// TIA Portal project "code_V15.1" (V15.1)

(* hardware
DEVICE "S7-1200 station_1"  S7-1200 Station
   slot 0: "Rack_0"  S7-1200 Rack  Rack  V1.0
   slot 1: "PLC_1"  CPU 1212C AC/DC/Rly  6ES7 212-1BE40-0XB0  V4.2
DEVICE "PC-System_1"  SIMATIC PC station
   slot 0: "SIMATIC PC station"  Rail  SIMATIC PC-Station  V1.0
      slot 125: "Stationmanager"  Station_Manager  V6.0.4
   slot 1: "HMI_RT_1"  WinCC RT Advanced  6AV2 104-0xxxx-xxxx  15.0.0.0
      slot 33792: "Host interface"  Host interface
   slot 2: "IE general_1"  IE General  IE_CP  V8.2.0
*)

// ===== PLC "PLC_1"  CPU 1212C AC/DC/Rly =====

VAR_GLOBAL   // PLC tag table "INPUT"
   "start" AT %M0.0 : Bool;
   "vatDo" AT %M0.1 : Bool;
   "vatXanh" AT %M0.2 : Bool;
   "CB1" AT %M0.3 : Bool;
   "reset" AT %M0.4 : Bool;
   "bd" AT %M0.5 : Bool;
END_VAR

VAR_GLOBAL   // PLC tag table "OUTPUT"
   "soVatDo" AT %MW100 : Int;
   "soVatXanh" AT %MW102 : Int;
   "vatDoDiChuyen" AT %MW104 : Int;
   "vatXanhDiChuyen" AT %MW106 : Int;
   "demmaudo" AT %MW116 : Int;
   "demmauxanh" AT %MW118 : Int;
END_VAR

VAR_GLOBAL   // PLC tag table "TG"
   "tg1" AT %M50.0 : Bool;
   "tg2" AT %M50.1 : Bool;
   "tg3" AT %M50.2 : Bool;
   "tg4" AT %M50.3 : Bool;
   "tg5" AT %M50.4 : Bool;
   "tg6" AT %M50.5 : Bool;
   "tg7" AT %M50.6 : Bool;
   "tg8" AT %M50.7 : Bool;
   "vatdodi" AT %M51.0 : Bool;
   "vatxanhdi" AT %M51.1 : Bool;
   "tg11" AT %M51.2 : Bool;
   "tg12" AT %M51.3 : Bool;
   "tg13" AT %M51.4 : Bool;
   "tg14" AT %M51.5 : Bool;
   "tg15" AT %M51.6 : Bool;
   "tg16" AT %M51.7 : Bool;
   "tg17" AT %M52.0 : Bool;
   "tg18" AT %Q0.0 : Bool;
   "tg19" AT %M52.2 : Bool;
   "tg20" AT %M52.3 : Bool;
   "tg21" AT %M52.4 : Bool;
   "tg22" AT %M52.5 : Bool;
   "tg23" AT %M52.6 : Bool;
   "tg24" AT %M52.7 : Bool;
   "tg25" AT %M53.0 : Bool;
   "TG_star" AT %M49.7 : Bool;
   "xung1" AT %M53.1 : Bool;
   "xung2" AT %M53.2 : Bool;
   "xung3" AT %M53.3 : Bool;
   "xung4" AT %M53.4 : Bool;
   "xung5" AT %M53.5 : Bool;
   "xung6" AT %M53.6 : Bool;
   "xung7" AT %M53.7 : Bool;
   "xung8" AT %M54.0 : Bool;
   "xung9" AT %M54.1 : Bool;
   "xung10" AT %M54.2 : Bool;
END_VAR

VAR_GLOBAL   // PLC tag table "TAYMAY"
   "tayKepDo" AT %M20.0 : Bool;
   "tayKepXanh" AT %M20.1 : Bool;
   "tayKepDo_diChuyenDi" AT %MW108 : Int;
   "tayKepDo_diChuyenVe" AT %MW110 : Int;
   "tayKepXanh_diChuyenDi" AT %MW112 : Int;
   "tayKepXanh_diChuyenVe" AT %MW114 : Int;
   "hienthitaybandau" AT %MW120 : Int;
END_VAR

// folder: System blocks/Program resources

DATA_BLOCK "time0"   // DB1
{ S7_Optimized_Access := 'TRUE' }
AUTHOR : Simatic
FAMILY : IEC
NAME : IEC_TMR
VERSION : 1.0
// stored: InstanceOfName IEC_TIMER
"IEC_TIMER"
BEGIN
END_DATA_BLOCK

DATA_BLOCK "time1"   // DB2
{ S7_Optimized_Access := 'TRUE' }
AUTHOR : Simatic
FAMILY : IEC
NAME : IEC_TMR
VERSION : 1.0
// stored: InstanceOfName IEC_TIMER
"IEC_TIMER"
BEGIN
END_DATA_BLOCK

DATA_BLOCK "time2"   // DB3
{ S7_Optimized_Access := 'TRUE' }
AUTHOR : Simatic
FAMILY : IEC
NAME : IEC_TMR
VERSION : 1.0
// stored: InstanceOfName IEC_TIMER
"IEC_TIMER"
BEGIN
END_DATA_BLOCK

DATA_BLOCK "time3"   // DB4
{ S7_Optimized_Access := 'TRUE' }
AUTHOR : Simatic
FAMILY : IEC
NAME : IEC_TMR
VERSION : 1.0
// stored: InstanceOfName IEC_TIMER
"IEC_TIMER"
BEGIN
END_DATA_BLOCK

DATA_BLOCK "IEC_Timer_0_DB"   // DB5
{ S7_Optimized_Access := 'TRUE' }
AUTHOR : Simatic
FAMILY : IEC
NAME : IEC_TMR
VERSION : 1.0
// stored: InstanceOfName IEC_TIMER
"IEC_TIMER"
BEGIN
END_DATA_BLOCK

DATA_BLOCK "IEC_Timer_0_DB_1"   // DB6
{ S7_Optimized_Access := 'TRUE' }
AUTHOR : Simatic
FAMILY : IEC
NAME : IEC_TMR
VERSION : 1.0
// stored: InstanceOfName IEC_TIMER
"IEC_TIMER"
BEGIN
END_DATA_BLOCK

DATA_BLOCK "time4"   // DB7
{ S7_Optimized_Access := 'TRUE' }
AUTHOR : Simatic
FAMILY : IEC
NAME : IEC_TMR
VERSION : 1.0
// stored: InstanceOfName IEC_TIMER
"IEC_TIMER"
BEGIN
END_DATA_BLOCK

DATA_BLOCK "time5"   // DB8
{ S7_Optimized_Access := 'TRUE' }
AUTHOR : Simatic
FAMILY : IEC
NAME : IEC_TMR
VERSION : 1.0
// stored: InstanceOfName IEC_TIMER
"IEC_TIMER"
BEGIN
END_DATA_BLOCK

// folder: (top level)

FUNCTION "simulation" : Void   // FC1, LAD
{ S7_Optimized_Access := 'TRUE' }
VERSION : 0.1
   VAR_TEMP   // added for the SCL form of the ladder/FBD networks
      _w1 : Bool;
   END_VAR
BEGIN

REGION Network 1
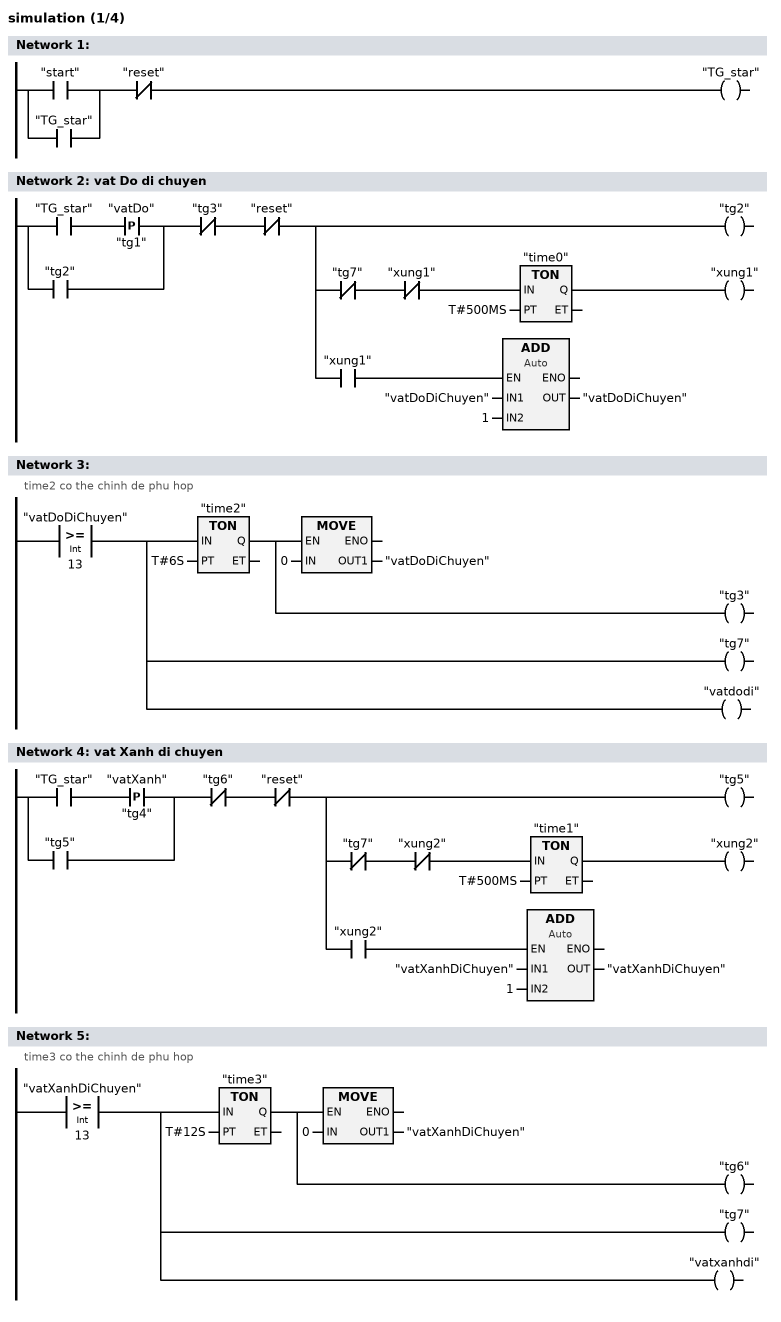
   RUNG wire#powerrail
      Contact( "start" )
      wire#w1
      I_Contact( "reset" )
      Coil( "TG_star" )
   END_RUNG
   RUNG wire#powerrail
      Contact( "TG_star" )
   END_RUNG wire#w1
   // the same network as SCL:
   "TG_star" := ("start" OR "TG_star") AND NOT "reset";
END_REGION

REGION Network 2: vat Do di chuyen
   #_w1 := "TG_star" AND "vatDo" AND NOT "tg1";   // rising edge of "vatDo"
   "tg1" := "vatDo";
   "tg2" := (#_w1 OR "tg2") AND NOT "tg3" AND NOT "reset";
   "time0".TON(IN := "tg2" AND NOT "tg7" AND NOT "xung1", PT := T#500MS);
   "xung1" := "time0".Q;
   IF "tg2" AND "xung1" THEN "vatDoDiChuyen" := "vatDoDiChuyen" + 1; END_IF;
END_REGION

REGION Network 3
   // time2 co the chinh de phu hop
   #_w1 := "vatDoDiChuyen" >= 13;
   "time2".TON(IN := #_w1, PT := T#6S);
   IF "time2".Q THEN "vatDoDiChuyen" := 0; END_IF;
   "tg3" := "time2".Q;
   "tg7" := #_w1;
   "vatdodi" := #_w1;
END_REGION

REGION Network 4: vat Xanh di chuyen
   #_w1 := "TG_star" AND "vatXanh" AND NOT "tg4";   // rising edge of "vatXanh"
   "tg4" := "vatXanh";
   "tg5" := (#_w1 OR "tg5") AND NOT "tg6" AND NOT "reset";
   "time1".TON(IN := "tg5" AND NOT "tg7" AND NOT "xung2", PT := T#500MS);
   "xung2" := "time1".Q;
   IF "tg5" AND "xung2" THEN "vatXanhDiChuyen" := "vatXanhDiChuyen" + 1; END_IF;
END_REGION

REGION Network 5
   // time3 co the chinh de phu hop
   #_w1 := "vatXanhDiChuyen" >= 13;
   "time3".TON(IN := #_w1, PT := T#12S);
   IF "time3".Q THEN "vatXanhDiChuyen" := 0; END_IF;
   "tg6" := "time3".Q;
   "tg7" := #_w1;
   "vatxanhdi" := #_w1;
END_REGION

REGION Network 6: canh tay gap vat mau do
   // di
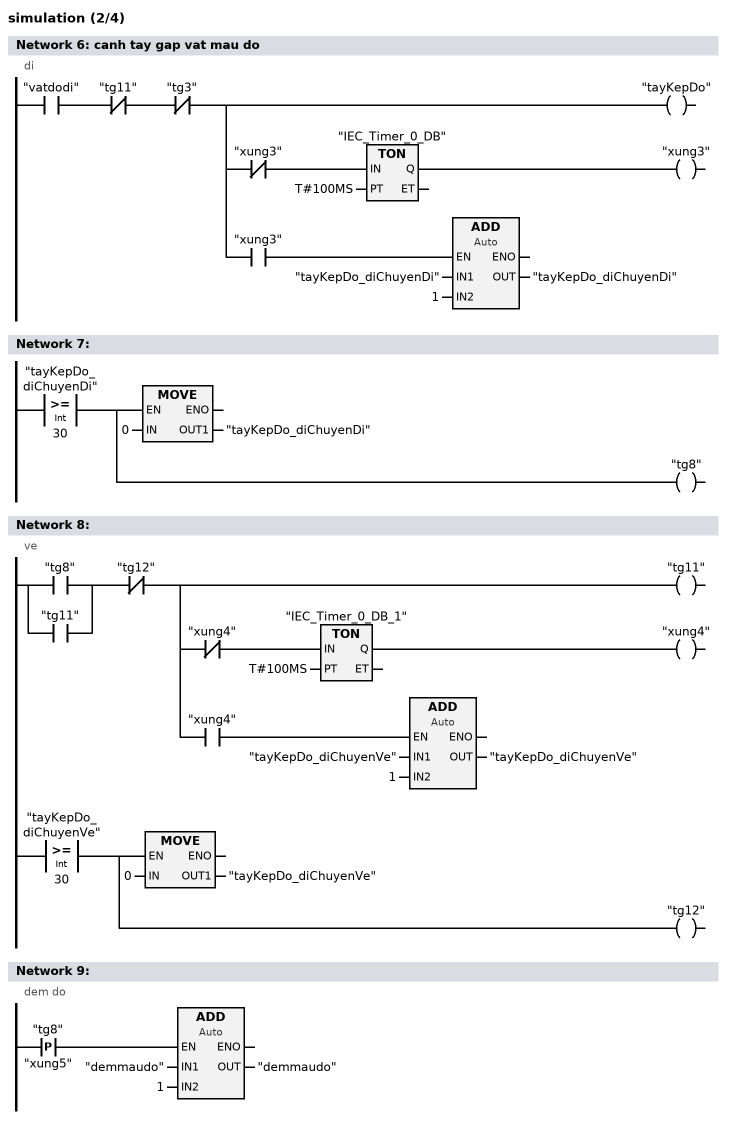
   "tayKepDo" := "vatdodi" AND NOT "tg11" AND NOT "tg3";
   "IEC_Timer_0_DB".TON(IN := "tayKepDo" AND NOT "xung3", PT := T#100MS);
   "xung3" := "IEC_Timer_0_DB".Q;
   IF "tayKepDo" AND "xung3" THEN "tayKepDo_diChuyenDi" := "tayKepDo_diChuyenDi" + 1; END_IF;
END_REGION

REGION Network 7
   RUNG wire#powerrail
      { S7_Templates := "SrcType := Int" } GE_Contact(in1 := "tayKepDo_diChuyenDi", in2 := 30)
      wire#w1
      Move(in := 0, out1 => "tayKepDo_diChuyenDi")
   END_RUNG
   RUNG wire#w1
      Coil( "tg8" )
   END_RUNG
   // the same network as SCL:
   #_w1 := "tayKepDo_diChuyenDi" >= 30;
   IF #_w1 THEN "tayKepDo_diChuyenDi" := 0; END_IF;
   "tg8" := #_w1;
END_REGION

REGION Network 8
   // ve
   "tg11" := ("tg8" OR "tg11") AND NOT "tg12";
   "IEC_Timer_0_DB_1".TON(IN := "tg11" AND NOT "xung4", PT := T#100MS);
   "xung4" := "IEC_Timer_0_DB_1".Q;
   IF "tg11" AND "xung4" THEN "tayKepDo_diChuyenVe" := "tayKepDo_diChuyenVe" + 1; END_IF;
   #_w1 := "tayKepDo_diChuyenVe" >= 30;
   IF #_w1 THEN "tayKepDo_diChuyenVe" := 0; END_IF;
   "tg12" := #_w1;
END_REGION

REGION Network 9
   // dem do
   RUNG wire#powerrail
      P_Contact(operand := "tg8", bit := "xung5")
      Add(in1 := "demmaudo", in2 := 1, out => "demmaudo")
   END_RUNG
   // the same network as SCL:
   #_w1 := "tg8" AND NOT "xung5";   // rising edge of "tg8"
   "xung5" := "tg8";
   IF #_w1 THEN "demmaudo" := "demmaudo" + 1; END_IF;
END_REGION

REGION Network 10: canh tay gap vat mau xanh
   // di
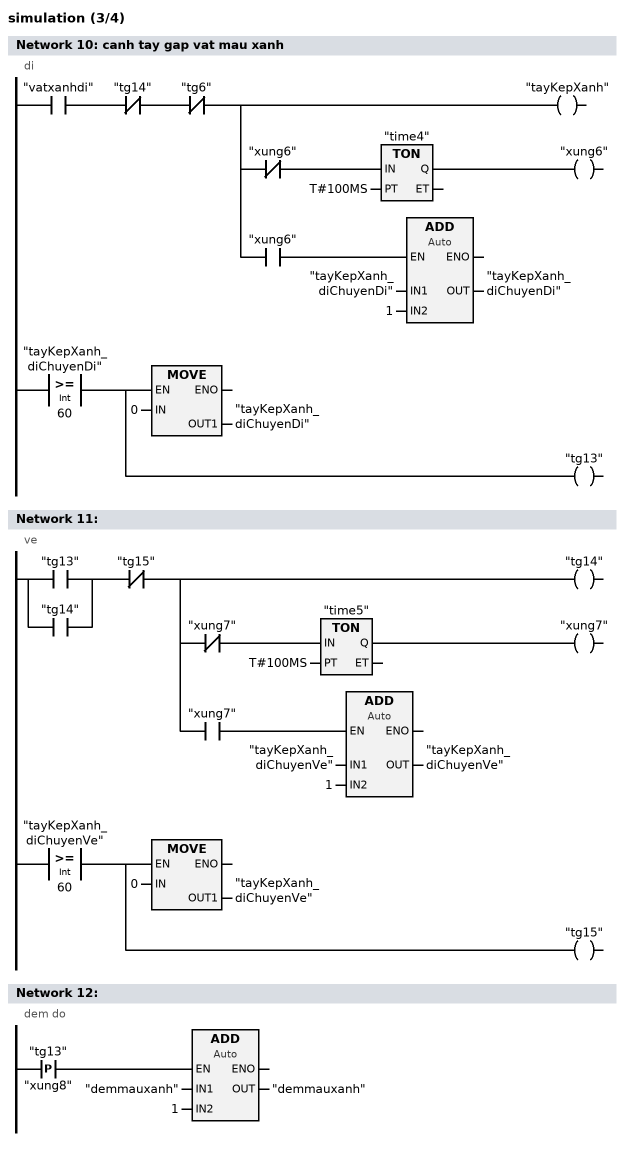
   "tayKepXanh" := "vatxanhdi" AND NOT "tg14" AND NOT "tg6";
   "time4".TON(IN := "tayKepXanh" AND NOT "xung6", PT := T#100MS);
   "xung6" := "time4".Q;
   IF "tayKepXanh" AND "xung6" THEN "tayKepXanh_diChuyenDi" := "tayKepXanh_diChuyenDi" + 1; END_IF;
   #_w1 := "tayKepXanh_diChuyenDi" >= 60;
   IF #_w1 THEN "tayKepXanh_diChuyenDi" := 0; END_IF;
   "tg13" := #_w1;
END_REGION

REGION Network 11
   // ve
   "tg14" := ("tg13" OR "tg14") AND NOT "tg15";
   "time5".TON(IN := "tg14" AND NOT "xung7", PT := T#100MS);
   "xung7" := "time5".Q;
   IF "tg14" AND "xung7" THEN "tayKepXanh_diChuyenVe" := "tayKepXanh_diChuyenVe" + 1; END_IF;
   #_w1 := "tayKepXanh_diChuyenVe" >= 60;
   IF #_w1 THEN "tayKepXanh_diChuyenVe" := 0; END_IF;
   "tg15" := #_w1;
END_REGION

REGION Network 12
   // dem do
   RUNG wire#powerrail
      P_Contact(operand := "tg13", bit := "xung8")
      Add(in1 := "demmauxanh", in2 := 1, out => "demmauxanh")
   END_RUNG
   // the same network as SCL:
   #_w1 := "tg13" AND NOT "xung8";   // rising edge of "tg13"
   "xung8" := "tg13";
   IF #_w1 THEN "demmauxanh" := "demmauxanh" + 1; END_IF;
END_REGION

REGION Network 13
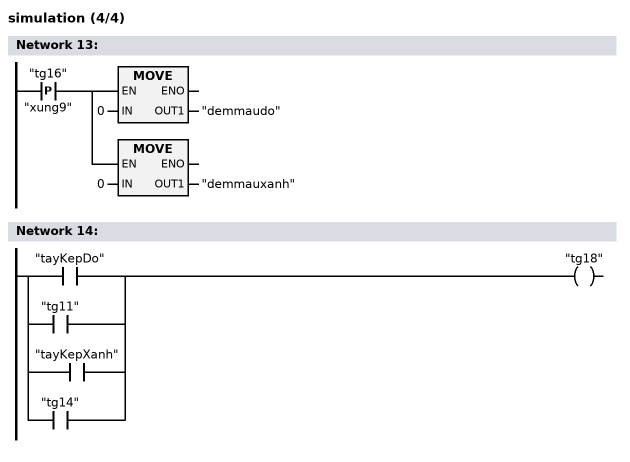
   RUNG wire#powerrail
      P_Contact(operand := "tg16", bit := "xung9")
      wire#w1
      Move(in := 0, out1 => "demmaudo")
   END_RUNG
   RUNG wire#w1
      Move(in := 0, out1 => "demmauxanh")
   END_RUNG
   // the same network as SCL:
   #_w1 := "tg16" AND NOT "xung9";   // rising edge of "tg16"
   "xung9" := "tg16";
   IF #_w1 THEN
       "demmaudo" := 0;
       "demmauxanh" := 0;
   END_IF;
END_REGION

REGION Network 14
   RUNG wire#powerrail
      Contact( "tayKepDo" )
      wire#w1
      Coil( "tg18" )
   END_RUNG
   RUNG wire#powerrail
      Contact( "tg11" )
   END_RUNG wire#w1
   RUNG wire#powerrail
      Contact( "tayKepXanh" )
   END_RUNG wire#w1
   RUNG wire#powerrail
      Contact( "tg14" )
   END_RUNG wire#w1
   // the same network as SCL:
   "tg18" := "tayKepDo" OR "tg11" OR "tayKepXanh" OR "tg14";
END_REGION
END_FUNCTION

ORGANIZATION_BLOCK "Main"   // OB1, LAD, ProgramCycle
TITLE = "Main Program Sweep (Cycle)"
{ S7_Optimized_Access := 'TRUE' }
VERSION : 0.1
   VAR_INPUT
      Initial_Call : Bool;   // Initial call of this OB
      Remanence : Bool;   // =True, if remanent data are available
   END_VAR
   VAR_TEMP   // added for the SCL form of the ladder/FBD networks
      _w1 : Bool;
      _w2 : Bool;
   END_VAR
BEGIN

REGION Network 1
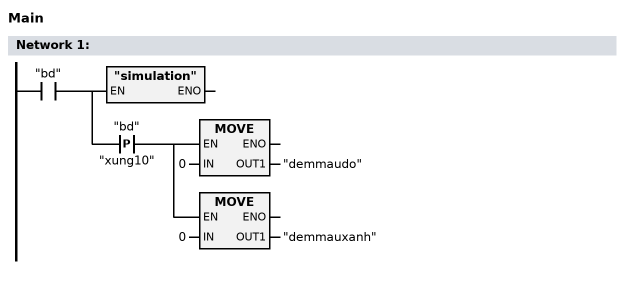
   RUNG wire#powerrail
      Contact( "bd" )
      wire#w1
      "simulation"()
   END_RUNG
   RUNG wire#w1
      P_Contact(operand := "bd", bit := "xung10")
      wire#w2
      Move(in := 0, out1 => "demmaudo")
   END_RUNG
   RUNG wire#w2
      Move(in := 0, out1 => "demmauxanh")
   END_RUNG
   // the same network as SCL:
   #_w1 := "bd";
   IF #_w1 THEN "simulation"(); END_IF;
   #_w2 := #_w1 AND "bd" AND NOT "xung10";   // rising edge of "bd"
   "xung10" := "bd";
   IF #_w2 THEN
       "demmaudo" := 0;
       "demmauxanh" := 0;
   END_IF;
END_REGION
END_ORGANIZATION_BLOCK

(* ===== HMI "HMI_RT_1" =====
system functions are stored by id; their names below are inferred from use
connection "HMI_Connection_1": ETHERNET, S7_1200_OMS

HMI tags "Default tag table"
   "start" : Bool = PLC start AT %M0.0, 1 s
   "reset" : Bool = PLC reset AT %M0.4, 1 s
   "vatDo" : Bool = PLC vatDo AT %M0.1, 1 s
   "vatXanh" : Bool = PLC vatXanh AT %M0.2, 1 s
   "simulation(1)" : Bool = PLC bd AT %M0.5, 1 s
   "vatDoDiChuyen" : Int = PLC vatDoDiChuyen AT %MW104, 1 s
   "vatXanhDiChuyen" : Int = PLC vatXanhDiChuyen AT %MW106, 1 s
   "anVatXanh" : Bool = PLC vatdodi AT %M51.0, 1 s
   "anVatDo" : Bool = PLC tg8 AT %M50.7, 1 s
   "tg7" : Bool = PLC tg7 AT %M50.6, 1 s
   "tayKepDo_diChuyenDi" : Int = PLC tayKepDo_diChuyenDi AT %MW108, 1 s
   "tayKepDo" : Bool = PLC tayKepDo AT %M20.0, 1 s
   "tg11" : Bool = PLC tg11 AT %M51.2, 1 s
   "tayKepDo_diChuyenVe" : Int = PLC tayKepDo_diChuyenVe AT %MW110, 1 s
   "time2_ET" : Time = PLC time2.ET, 1 s
   "tayKepXanh_diChuyenDi" : Int = PLC tayKepXanh_diChuyenDi AT %MW112, 1 s
   "tg16" : Bool = PLC tg16 AT %M51.7, 1 s
   "tg14" : Bool = PLC tg14 AT %M51.5, 1 s
   "tayKepXanh_diChuyenVe" : Int = PLC tayKepXanh_diChuyenVe AT %MW114, 1 s
   "tayKepXanh" : Bool = PLC tayKepXanh AT %M20.1, 1 s
   "demmaudo" : Int = PLC demmaudo AT %MW116, 1 s
   "demmauxanh" : Int = PLC demmauxanh AT %MW118, 1 s
   "tg18" : Bool = PLC tg18 AT %Q0.0, 1 s
   "hienthitaybandau" : Int = PLC hienthitaybandau AT %MW120, 1 s

screen "Screen_1" 1024x768
   Button "Button_1" at 31,100 size 96x32; TextOff 'START'
      on Press: SetBit("start")
      on Release: ResetBit("start")
      Appearance <- "start"
   Button "Button_3" at 158,99 size 96x32; TextOff 'RED'
      on Press: SetBit("vatDo")
      on Release: ResetBit("vatDo")
      Appearance <- "vatDo"
   Button "Button_4" at 157,154 size 96x32; TextOff 'GREEN'
      on Press: SetBit("vatXanh")
      on Release: ResetBit("vatXanh")
      Appearance <- "vatXanh"
   Switch "Switch_1" at 71,23 size 143x49; CaptionText 'SIMULATION'; TextOff 'OFF'; TextOn 'ON'
      on SwitchOn: SetBit("simulation(1)")
      on SwitchOff: ResetBit("simulation(1)")
   SymbolLibrary "Symbol library_1" at 81,355 size 279x58
   Rectangle "Rectangle_2" at 71,337 size 38x37
      HorizontalMovement <- "vatDoDiChuyen"
      Visibility <- "vatDoDiChuyen"
   SymbolLibrary "Symbol library_2" at 304,425 size 20x62
      Appearance <- "tg7"
   Rectangle "Rectangle_1" at 60,337 size 38x37
      HorizontalMovement <- "vatXanhDiChuyen"
      Visibility <- "vatXanhDiChuyen"
   SymbolLibrary "Symbol library_3" at 466,357 size 121x79
   Rectangle "Rectangle_9" at 517,171 size 29x37
      Appearance <- "tayKepDo"
   Rectangle "Rectangle_10" at 733,171 size 29x37
      Appearance <- "tayKepXanh"
   SymbolLibrary "Symbol library_4" at 690,355 size 112x79
   TextField "Text field_1" at 502,403 size 36x22; Text 'RED'
   TextField "Text field_2" at 710,403 size 56x22; Text 'GREED'
   Group "Group_2" at 502,223 size 59x111
   Group "Group_1" at 286,223 size 59x117
   Button "Button_5" at 31,154 size 96x32; TextOff 'reset'
      on Press: SetBit("tg16")
      on Release: ResetBit("tg16")
      Appearance <- "tg16"
   Group "Group_4" at 719,223 size 59x111
   IOField "I/O field_1" at 480,451 size 96x32; FormatPattern s99999
      ProcessValue <- "demmaudo"
   IOField "I/O field_2" at 700,451 size 96x32; FormatPattern s99999
      ProcessValue <- "demmauxanh"
   Group "Group_3" at 286,223 size 59x117
   Group "Group" at 286,223 size 59x111
   Rectangle "Rectangle_6" at 286,303 size 11x31
      Visibility <- "tg18"
   Rectangle "Rectangle_4" at 303,223 size 23x69
      Visibility <- "tg18"
   Rectangle "Rectangle_5" at 286,292 size 59x11
      Visibility <- "tg18"
   Rectangle "Rectangle_7" at 334,303 size 11x31
      Visibility <- "tg18"
   Rectangle "Rectangle_17" at 502,303 size 11x31
      Visibility <- "tg11"
      HorizontalMovement <- "tayKepDo_diChuyenVe"
   Rectangle "Rectangle_16" at 502,292 size 59x11
      Visibility <- "tg11"
      HorizontalMovement <- "tayKepDo_diChuyenVe"
   Rectangle "Rectangle_18" at 550,303 size 11x31
      Visibility <- "tg11"
      HorizontalMovement <- "tayKepDo_diChuyenVe"
   Rectangle "Rectangle_15" at 519,223 size 23x69
      Visibility <- "tg11"
      HorizontalMovement <- "tayKepDo_diChuyenVe"
   Rectangle "Rectangle_22" at 303,223 size 23x69
      HorizontalMovement <- "tayKepXanh_diChuyenDi"
      Visibility <- "tayKepXanh_diChuyenDi"
   Rectangle "Rectangle_20" at 334,303 size 11x31
      HorizontalMovement <- "tayKepXanh_diChuyenDi"
      Visibility <- "tayKepXanh_diChuyenDi"
   Rectangle "Rectangle_21" at 286,292 size 59x11
      HorizontalMovement <- "tayKepXanh_diChuyenDi"
      Visibility <- "tayKepXanh_diChuyenDi"
   Rectangle "Rectangle_19" at 286,303 size 11x31
      HorizontalMovement <- "tayKepXanh_diChuyenDi"
      Visibility <- "tayKepXanh_diChuyenDi"
   Rectangle "Rectangle_24" at 297,303 size 38x37
      HorizontalMovement <- "tayKepXanh_diChuyenDi"
      Visibility <- "tayKepXanh_diChuyenDi"
   Rectangle "Rectangle_23" at 297,303 size 38x37
      Visibility <- "tayKepDo_diChuyenDi"
      HorizontalMovement <- "tayKepDo_diChuyenDi"
   Rectangle "Rectangle_13" at 286,303 size 11x31
      HorizontalMovement <- "tayKepDo_diChuyenDi"
      Visibility <- "tayKepDo_diChuyenDi"
   Rectangle "Rectangle_12" at 286,292 size 59x11
      HorizontalMovement <- "tayKepDo_diChuyenDi"
      Visibility <- "tayKepDo_diChuyenDi"
   Rectangle "Rectangle_14" at 303,223 size 23x69
      HorizontalMovement <- "tayKepDo_diChuyenDi"
      Visibility <- "tayKepDo_diChuyenDi"
   Rectangle "Rectangle_11" at 334,303 size 11x31
      HorizontalMovement <- "tayKepDo_diChuyenDi"
      Visibility <- "tayKepDo_diChuyenDi"
   Rectangle "Rectangle_27" at 767,303 size 11x31
      Visibility <- "tg14"
      HorizontalMovement <- "tayKepXanh_diChuyenVe"
   Rectangle "Rectangle_25" at 719,303 size 11x31
      Visibility <- "tg14"
      HorizontalMovement <- "tayKepXanh_diChuyenVe"
   Rectangle "Rectangle_26" at 719,292 size 59x11
      Visibility <- "tg14"
      HorizontalMovement <- "tayKepXanh_diChuyenVe"
   Rectangle "Rectangle_28" at 736,223 size 23x69
      Visibility <- "tg14"
      HorizontalMovement <- "tayKepXanh_diChuyenVe"
*)